PROGRAM storage
VAR
END_VAR

bStorage :=UDINT_TO_BOOL(PositionTrigger[1].CurrentMover.AxisReference.NcToPlc.AxisId MOD 2);
				IF bStorage THEN
					IF bStorage THEN
						Station[0].UnregisterMover(PositionTrigger[1].CurrentMover);
						PositionTrigger[1].CurrentMover.MoveToStation(Station[1]);
					END_IF
				END_IF

END_PROGRAM

(* stored: Version 1.1.0.1, ProductVersion 3.1.4024.9
   POU storage: Id {14c4a04e-619b-4c9d-845c-f616f2e44d96}, SpecialFunc None *)
